{attribute 'GeneratedUsingTerminal: EL1809-0000-0018'}
{attribute addProperty BoxType "EL1809-0000-0018"}
{attribute addProperty Id "StateAT %I*UINT2"}
{attribute addProperty CRC "1863965483"}
{attribute addProperty Size "2"}
TYPE InfoData_6F19DB2B :
STRUCT
	{attribute addProperty Name "State"}
	State AT %I* : UINT;
END_STRUCT
END_TYPE

(* stored: Version 1.2.0.0, ProductVersion 3.1.4024.9
   DUT InfoData_6F19DB2B: Id {f3c8dc9c-236a-08f8-2a89-96d1caf15302} *)
